% RSLogix 500 project PROJECT1.RSS, saved by version 8.30.00.16 %
PROJECT "UNTITLED"    % processor: Bul.1763 MicroLogix 1100 Series B %

PROGRAM FILES
  LAD 2 "MAIN"  4 rungs
  LAD 3 "DI/DO"  5 rungs
  LAD 4 "CONTROL"  3 rungs

DATA FILES
  O0 OUTPUT  5 elements
  I1 INPUT  7 elements
  S2 STATUS  66 elements
  B3 BINARY  1 elements
  T4 TIMER  1 elements
  C5 COUNTER  1 elements
  R6 CONTROL  1 elements
  N7 INTEGER  1 elements
  F8 FLOAT  1 elements

LADDER 2 "MAIN"
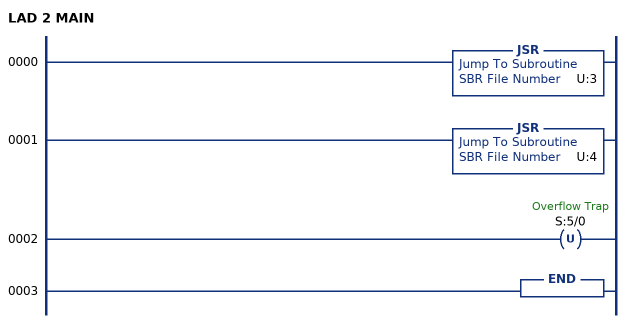
% Rung: 0 %
SOR JSR U:3 EOR
% Rung: 1 %
SOR JSR U:4 EOR
% Rung: 2 %
SOR OTU S:5/0 EOR
%   S:5/0  "Overflow Trap" %
% Rung: 3 %
SOR END EOR

LADDER 3 "DI/DO"
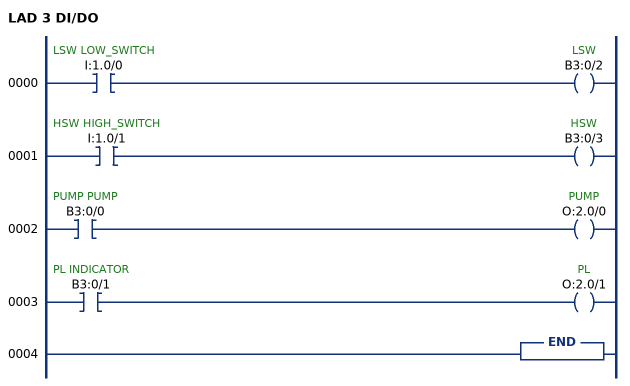
% Rung: 0 %
SOR XIC I:1.0/0 OTE B3:0/2 EOR
%   I:1.0/0  LOW_SWITCH  "LSW" %
%   B3:0/2  "LSW" %
% Rung: 1 %
SOR XIC I:1.0/1 OTE B3:0/3 EOR
%   I:1.0/1  HIGH_SWITCH  "HSW" %
%   B3:0/3  "HSW" %
% Rung: 2 %
SOR XIC B3:0/0 OTE O:2.0/0 EOR
%   B3:0/0  PUMP  "PUMP" %
%   O:2.0/0  "PUMP" %
% Rung: 3 %
SOR XIC B3:0/1 OTE O:2.0/1 EOR
%   B3:0/1  INDICATOR  "PL" %
%   O:2.0/1  "PL" %
% Rung: 4 %
SOR END EOR

LADDER 4 "CONTROL"
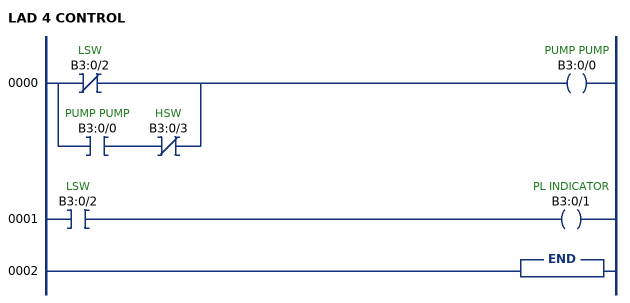
% Rung: 0 %
SOR BST XIO B3:0/2 NXB XIC B3:0/0 XIO B3:0/3 BND OTE B3:0/0 EOR
%   B3:0/2  "LSW" %
%   B3:0/0  PUMP  "PUMP" %
%   B3:0/3  "HSW" %
% Rung: 1 %
SOR XIC B3:0/2 OTE B3:0/1 EOR
%   B3:0/2  "LSW" %
%   B3:0/1  INDICATOR  "PL" %
% Rung: 2 %
SOR END EOR

OTHER DOCUMENTED ADDRESSES
  O:2.0/2  "PUMP"
  O:2.0/3  "PL"
